// TIA Portal V17 export
// export: Created 2023-04-04T13:27:28.3302551Z, ExportSetting WithDefaults, DisplayName Totally Integrated Automation Portal, DisplayVersion V17, DisplayName TIA Portal Openness, DisplayVersion V17, DisplayName TIA Portal Version Control Interface, DisplayVersion V17, DisplayName STEP 7 Professional, DisplayVersion V17, DisplayName STEP 7 Safety, DisplayVersion V17, DisplayName WinCC Advanced, DisplayVersion V17
DATA_BLOCK "gtyp_Interface_TXT_Controler"   // DB40
{ S7_Optimized_Access := 'TRUE' }
VERSION : 0.1
// stored: AutoNumber true, DBAccessibleFromOPCUA true, DBAccessibleFromWebserver true, InstanceOfName typ_MQTT_Interface_TXT_Controller, InstanceOfType UDT, IsOnlyStoredInLoadMemory false, IsWriteProtectedInAS false
"typ_MQTT_Interface_TXT_Controller"
   // VAR
   //    Subscribe { S7_SetPoint := 'True'} : "typ_MQTT_Interface_TXT_Controler_Subscribe";
   //    Publish { S7_SetPoint := 'True'} : "typ_MQTT_ Interface_TXT_Controler_Publish";
   // END_VAR
BEGIN
END_DATA_BLOCK
